Fanuc KAREL source: kt00823.KL

-- PROVISIONAL review KL for V770-1; original PC SHA256 57902589ea0bbc98eb3332da2169e7e2f3988dc0ee07c69eaf3c9c9198a3c967
-- Incomplete behavior may be omitted. Consult companion uncertainty JSON. Do not deploy.
PROGRAM KT00823
%NOLOCKGROUP
VAR
  R1 : REAL
  R2 : REAL
  OUT : REAL
BEGIN
  -- UNRESOLVED_PC offsets 5-16; opcodes 2E,23
  -- UNRESOLVED_PC offsets 21-32; opcodes 2E,23
  -- UNRESOLVED_PC offsets 37-48; opcodes 2E,23
  -- UNRESOLVED_PC offsets 53-64; opcodes 2E,23
  -- UNRESOLVED_PC offsets 69-84; opcodes 27,22,76,23
  -- UNRESOLVED_PC offsets 89-93; opcodes 7F
END KT00823
